{attribute 'GeneratedUsingTerminal: CU1128-0000-0001'}
{attribute addProperty BoxType "CU1128-0000-0001"}
{attribute addProperty Id "A_0006_CU1128_0000_0002A_0006_CU1128_0000_0002_812875A084A_0005_CU1128_0000_0001_2_CU1128_BCU1128_1FC0878B2A_0005_CU1128_0000_0001_3_CU1128_CCU1128_1FC0878B2"}
{attribute addProperty CRC "1940734460"}
{attribute addProperty Size "88"}
TYPE A_0005_CU1128_0000_0001_73AD41FC EXTENDS CU1128_1FC0878B :
STRUCT
	{attribute addProperty Name "A_0006_CU1128_0000_0002"}
	{attribute addProperty PreviousPort "A_0005(CU1128-0000-0001) : D"}
	A_0006_CU1128_0000_0002 : A_0006_CU1128_0000_0002_812875A0;
	{attribute addProperty Name "A_0005_CU1128_0000_0001_2_CU1128_B"}
	{attribute addProperty PreviousPort "A_0005(CU1128-0000-0001) : C"}
	A_0005_CU1128_0000_0001_2_CU1128_B : CU1128_1FC0878B;
	{attribute addProperty Name "A_0005_CU1128_0000_0001_3_CU1128_C"}
	{attribute addProperty PreviousPort "A_0005(CU1128-0000-0001)_2 (CU1128-B) : C"}
	A_0005_CU1128_0000_0001_3_CU1128_C : CU1128_1FC0878B;
END_STRUCT
END_TYPE

(* stored: Version 1.2.0.0, ProductVersion 3.1.4024.9
   DUT A_0005_CU1128_0000_0001_73AD41FC: Id {f79013cf-8407-43e1-a901-1da727c89879} *)
